TYPE PiperImplements :
STRUCT
	aborting : BOOL;
	booting : BOOL;
	clearing : BOOL;
	completing : BOOL;
	executing : BOOL;
	holding : BOOL;
	resetting : BOOL;
	starting : BOOL;
	stopping : BOOL;
	suspending : BOOL;
	unholding : BOOL;
	unsuspending : BOOL;
END_STRUCT
END_TYPE

(* stored: Version 1.1.0.1, ProductVersion 3.1.4024.12
   DUT PiperImplements: Id {2b51da57-a32f-49e3-8800-6b62ef18d8cd} *)
